ABB RAPID module: Wizard.modx

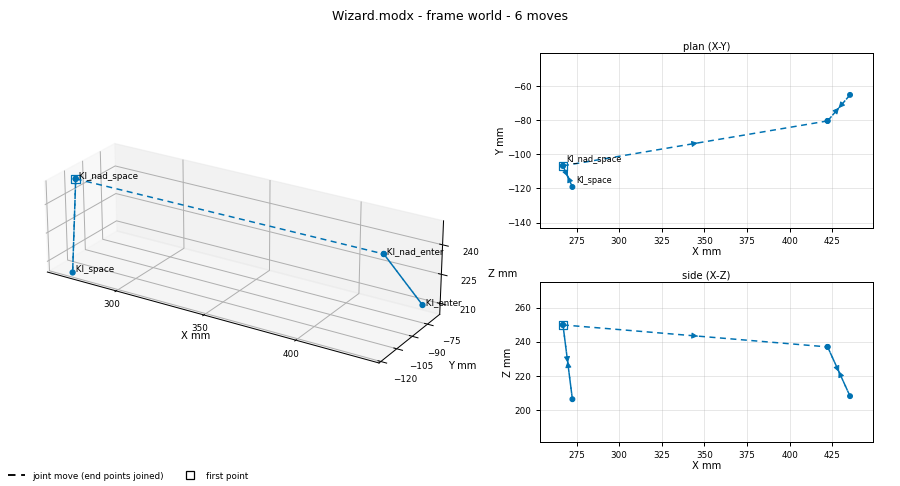
[picture p0: tool path of Wizard.modx in frame world, 6 of 6 moves have a stored position in this frame; points joined in program order, loops and branches not executed]
MODULE Wizard
PERS robtarget Location5:=[[-45.3218955993652, 414.107299804688, 542.560546875], [0.0331718660891056, 0.974595308303833, 0.220419079065323, 0.0218859035521746], [1, -1, -2, 0], [9000000000, 9000000000, 9000000000, 9000000000, 9000000000, 9000000000]];
PERS robtarget Location6:=[[-42.930736541748, 416.871459960938, 368.191131591797], [0.0221891868859529, 0.973919808864594, 0.225001737475395, 0.0190272349864244], [1, -1, -2, 0], [9000000000, 9000000000, 9000000000, 9000000000, 9000000000, 9000000000]];
PERS robtarget Location7:=[[-34.9866142272949, 458.268798828125, 584.186340332031], [0.00795904919505119, -0.978147804737091, -0.205494686961174, -0.0305846277624369], [1, -1, -2, 0], [9000000000, 9000000000, 9000000000, 9000000000, 9000000000, 9000000000]];
PERS robtarget Kl_space:=[[272.546997070313, -119.175819396973, 206.432632446289], [0.074522770941257, -0.494850546121597, -0.862464487552643, -0.075659230351448], [-1, 0, 0, 0], [9000000000, 9000000000, 9000000000, 9000000000, 9000000000, 9000000000]];
PERS robtarget Location8:=[[145.745910644531, 420.857421875, 492.48779296875], [0.0239510629326105, -0.999478936195374, 0.0202637929469347, 0.00758857233449817], [0, 0, -2, 0], [9000000000, 9000000000, 9000000000, 9000000000, 9000000000, 9000000000]];
PERS robtarget Location9:=[[-560.7, 509.56, 592.15], [0.00123678, -0.378767, 0.925393, 0.0135282], [1, -1, 1, 0], [9000000000, 9000000000, 9000000000, 9000000000, 9000000000, 9000000000]];
PERS robtarget Kl_enter:=[[435.378234863281, -65.1502075195313, 208.231979370117], [0.071741580963135, -0.797700226306915, -0.597699582576752, -0.0358140096068382], [-1, 0, 0, 0], [9000000000, 9000000000, 9000000000, 9000000000, 9000000000, 9000000000]];
PERS robtarget Location10:=[[613.03, 509.55, 592.16], [0.00125397, -0.378757, 0.925396, 0.0135404], [0, 0, -1, 0], [9000000000, 9000000000, 9000000000, 9000000000, 9000000000, 9000000000]];
PERS robtarget Location11:=[[60.7467308044434, 465.576812744141, 491.8779296875], [0.00205219932831824, -0.387099027633667, 0.921912610530853, 0.0150760682299733], [0, 0, 0, 0], [9000000000, 9000000000, 9000000000, 9000000000, 9000000000, 9000000000]];
PERS robtarget Location12:=[[60.7467498779297, 465.576934814453, 491.878173828125], [0.00205230480059981, -0.387099027633667, 0.921912610530853, 0.0150762461125851], [0, 0, 0, 0], [9000000000, 9000000000, 9000000000, 9000000000, 9000000000, 9000000000]];
PERS robtarget Location13:=[[41.1625862121582, 462.905975341797, 470.445495605469], [0.00223985756747425, -0.386858403682709, 0.922010123729706, 0.0152596672996879], [0, 0, 0, 0], [9000000000, 9000000000, 9000000000, 9000000000, 9000000000, 9000000000]];
PERS robtarget Kl_nad_space:=[[267.017120361328, -106.753517150879, 250.01481628418], [0.0316353738307953, -0.480643182992935, -0.872156977653503, -0.085577867925167], [-1, 0, 0, 0], [9000000000, 9000000000, 9000000000, 9000000000, 9000000000, 9000000000]];
PERS robtarget Location1:=[[141.020217895508, 436.321899414063, 575.21875], [0.017813965678215, 0.999827980995178, -0.000279141531791538, -0.0051563223823905], [0, -1, -2, 0], [9000000000, 9000000000, 9000000000, 9000000000, 9000000000, 9000000000]];
PERS robtarget Location2:=[[508.657287597656, 345.39111328125, 565.002990722656], [0.027114637196064, 0.945273578166962, -0.324619859457016, -0.018564136698842], [0, -1, -2, 0], [9000000000, 9000000000, 9000000000, 9000000000, 9000000000, 9000000000]];
PERS robtarget Location3:=[[138.697784423828, 217.932708740234, 413.045196533203], [0.07676836848259, 0.98807281255722, -0.127942427992821, -0.038071520626545], [0, 0, -2, 0], [9000000000, 9000000000, 9000000000, 9000000000, 9000000000, 9000000000]];
PERS robtarget Location4:=[[-51.5362167358398, 430.496246337891, 337.229919433594], [0.0170931983739138, -0.979323327541351, -0.201356798410416, 0.0094364807009697], [1, 0, -2, 0], [9000000000, 9000000000, 9000000000, 9000000000, 9000000000, 9000000000]];
PERS robtarget Kl_nad_enter:=[[422.22607421875, -80.4220809936523, 237.11946105957], [0.095908030867577, -0.757424414157867, -0.637956261634827, -0.100606605410576], [-1, 0, 0, 0], [9000000000, 9000000000, 9000000000, 9000000000, 9000000000, 9000000000]];
	PROC main()
SetDO ABB_Local_IO_0_DO1, 1;
MoveJ Kl_nad_space, v1000, fine, tool0;
MoveJ Kl_space, v1000, fine, tool0;
MoveJ Kl_nad_space, v1000, fine, tool0;
MoveJ Kl_nad_enter, v1000, fine, tool0;
MoveJ Kl_enter, v1000, fine, tool0;
MoveJ Kl_nad_enter, v1000, fine, tool0;
	ENDPROC
ENDMODULE
